TYPE ST_AnimationScaling :
STRUCT
	fPistonScale : LREAL := 200;
	fBoomScale : LREAL := 2;
END_STRUCT
END_TYPE

(* stored: Version 1.1.0.1, ProductVersion 3.1.4024.10
   DUT ST_AnimationScaling: Id {c85ff27b-304d-4688-9966-8b751276c145} *)
